// TwinCAT 3 PLC project EcLib
// ProgramVersion: 3.1.4023.0
// libraries:
//   Tc2_Standard, * (Beckhoff Automation GmbH)
//   Tc2_System, * (Beckhoff Automation GmbH)
//   Tc3_Module, * (Beckhoff Automation GmbH)
// project tree:
//   / PlcTask.TcTTO
//   POUs/ MAIN.TcPOU
//   Tasks/ EcMasterConfDevices.TcPOU, EcMasterDeviceCount.TcPOU, EcMasterDeviceState.TcPOU, EcMasterFrameCount.TcPOU, EcMasterFrameStats.TcPOU, EcMasterGetAbnortalStateChange.TcPOU, EcMasterGetDeviceCRC.TcPOU, EcMasterGetDeviceId.TcPOU, EcMasterGetDeviceState.TcPOU, EcMasterProtocolError.TcPOU, EcMasterScanDevices.TcPOU, EcMasterState.TcPOU, IEcTask.TcIO, ITask.TcIO

CONFIGURATION EcLib
    RESOURCE PLC ON TwinCAT3
        TASK PlcTask(INTERVAL := T#10ms, PRIORITY := 20);
        PROGRAM MAIN WITH PlcTask : MAIN;
    END_RESOURCE
END_CONFIGURATION

// ---- Tasks/IEcTask.TcIO
INTERFACE IEcTask EXTENDS ITask

PROPERTY NetID : amsnetid
GET
END_GET
SET
END_SET
END_PROPERTY

END_INTERFACE

// ---- Tasks/ITask.TcIO
INTERFACE ITask

METHOD Abort : BOOL
VAR_INPUT
END_VAR
END_METHOD

PROPERTY Busy : bool
GET
END_GET
END_PROPERTY

PROPERTY Done : bool
GET
END_GET
END_PROPERTY

PROPERTY Error : bool
GET
END_GET
END_PROPERTY

METHOD Execute : BOOL
VAR_INPUT
END_VAR
END_METHOD

END_INTERFACE

// ---- POUs/MAIN.TcPOU
PROGRAM MAIN
VAR
END_VAR

END_PROGRAM

// ---- Tasks/EcMasterConfDevices.TcPOU
FUNCTION_BLOCK EcMasterConfDevices IMPLEMENTS IEcTask
VAR_INPUT
END_VAR
VAR_OUTPUT
END_VAR
VAR
	iState : INT;
	masterConfDevices : Tc2_EtherCAT.FB_EcGetConfSlaves;
	_confDevices : ARRAY[0..Tc2_EtherCAT.EC_MAX_SLAVES] OF Tc2_EtherCAT.ST_EcSlaveConfigData;
	_execute: BOOL;
	_done: BOOL;
	_busy: BOOL;	
	_error: BOOL;
	_netId: AMSNETID;
END_VAR

CASE iState OF
	0:
		IF _execute THEN
			_done := FALSE;
			_busy := TRUE;
			_error := FALSE;
			masterConfDevices.bExecute := TRUE;
			IF masterConfDevices.bBusy THEN
				iState := 10;
				_execute := FALSE;
			END_IF
		END_IF
	10:
		IF NOT masterConfDevices.bBusy THEN
			IF NOT masterConfDevices.bError THEN
				_done := TRUE;
			ELSE
				_error := TRUE;
			END_IF
			_busy := FALSE;
			masterConfDevices.bExecute := FALSE;
			iState := 0;
		END_IF
END_CASE

masterConfDevices(sNetId := Tc2_System.F_CreateAmsNetId(nIds := NetId), 
					pArrEcConfSlaveInfo := ADR(_confDevices), 
					cbBufLen := SIZEOF(_confDevices));

{warning 'add method implementation '}
METHOD Abort : BOOL
masterConfDevices.bExecute := FALSE;
_busy := FALSE;
_execute := FALSE;
Abort := TRUE;
iState := 0;
END_METHOD

{warning 'add property implementation'}
PROPERTY Busy : BOOL
GET
Busy := _busy;
END_GET
END_PROPERTY

PROPERTY ConfiguredDevices : reference to array[0..Ec_Max_slaves] of St_ecslaveconfigdata
GET
ConfiguredDevices REF= _confDevices;
END_GET
END_PROPERTY

{warning 'add property implementation'}
PROPERTY Done : BOOL
GET
Done := _done;
END_GET
END_PROPERTY

{warning 'add property implementation'}
PROPERTY Error : BOOL
GET
Error := _error;
END_GET
END_PROPERTY

{warning 'add method implementation '}
METHOD Execute : BOOL
IF NOT masterConfDevices.bBusy THEN
	Execute := _execute := true;
END_IF
END_METHOD

{warning 'add property implementation'}
PROPERTY NetID : amsnetid
GET
NetID := _netId;
END_GET
SET
_netId := NetID;
END_SET
END_PROPERTY

PROPERTY NumberConfDevices : udint
GET
NumberConfDevices := masterConfDevices.nSlaves;
END_GET
END_PROPERTY

END_FUNCTION_BLOCK

// ---- Tasks/EcMasterDeviceCount.TcPOU
FUNCTION_BLOCK PUBLIC EcMasterDeviceCount IMPLEMENTS IEcTask
VAR_INPUT
END_VAR
VAR_OUTPUT
END_VAR
VAR
	iState : INT;
	masterDeviceCount : Tc2_EtherCAT.FB_EcGetSlaveCount;
	_execute: BOOL;
	_done: BOOL;
	_busy: BOOL;
	_error: BOOL;
	_netId: AMSNETID;
END_VAR

CASE iState OF
	0:
		IF _execute THEN
			_done := FALSE;
			_busy := TRUE;
			_error := FALSE;
			masterDeviceCount.bExecute := TRUE;
			IF masterDeviceCount.bBusy THEN
				iState := 10;
				_execute := false;
			END_IF
		END_IF
	10:
		IF NOT masterDeviceCount.bBusy THEN
			IF NOT masterDeviceCount.bError THEN
				_done := TRUE;
			ELSE
				_error := TRUE;
			END_IF
			_busy := FALSE;
			masterDeviceCount.bExecute := FALSE;
			iState := 0;
		END_IF
END_CASE

masterDeviceCount(sNetId := Tc2_System.F_CreateAmsNetId(nIds := NetId));

{warning 'add method implementation '}
METHOD Abort : BOOL
masterDeviceCount.bExecute := FALSE;
_busy := FALSE;
_execute := FALSE;
Abort := TRUE;
iState := 0;
END_METHOD

{warning 'add property implementation'}
PROPERTY Busy : BOOL
GET
Busy := _busy;
END_GET
END_PROPERTY

{warning 'add property implementation'}
PROPERTY Done : BOOL
GET
Done := _done;
END_GET
END_PROPERTY

{warning 'add property implementation'}
PROPERTY Error : BOOL
GET
Error := _error;
END_GET
END_PROPERTY

METHOD Execute : BOOL
VAR_INPUT
END_VAR
IF NOT Busy THEN
	Execute := _execute := TRUE;
END_IF
END_METHOD

{warning 'add property implementation'}
PROPERTY NetID : amsnetid
GET
NetID := _netId;
END_GET
SET
_netId := NetID;
END_SET
END_PROPERTY

PROPERTY NumberDevices : uint
GET
NumberDevices := masterDeviceCount.nSlaves;
END_GET
END_PROPERTY

END_FUNCTION_BLOCK

// ---- Tasks/EcMasterDeviceState.TcPOU
FUNCTION_BLOCK EcMasterDeviceState IMPLEMENTS IEcTask
VAR_INPUT
END_VAR
VAR_OUTPUT
END_VAR
VAR
	iState : INT;
	masterDeviceState : Tc2_EtherCAT.FB_EcGetMasterDevState;
	_execute: BOOL;
	_done: BOOL;
	_busy: BOOL;
	_error: BOOL;
	_netId: AMSNETID;
END_VAR

CASE iState OF
	0:
		IF _execute THEN
			_done := FALSE;
			_busy := TRUE;
			_error := FALSE;
			masterDeviceState.bExecute := TRUE;
			IF masterDeviceState.bBusy THEN
				iState := 10;
				_execute := false;
			END_IF
		END_IF
	10:
		IF NOT masterDeviceState.bBusy THEN
			IF NOT masterDeviceState.bError THEN
				_done := TRUE;
			ELSE
				_error := TRUE;
			END_IF
			_busy := FALSE;
			masterDeviceState.bExecute := FALSE;
			iState := 0;
		END_IF
END_CASE

masterDeviceState(sNetId := Tc2_System.F_CreateAmsNetId(nIds := NetId));

{warning 'add method implementation '}
METHOD Abort : BOOL
masterDeviceState.bExecute := FALSE;
_busy := FALSE;
_execute := FALSE;
Abort := TRUE;
iState := 0;
END_METHOD

{warning 'add property implementation'}
PROPERTY Busy : BOOL
GET
Busy := _busy;
END_GET
END_PROPERTY

{warning 'add property implementation'}
PROPERTY Done : BOOL
GET
Done := _done;
END_GET
END_PROPERTY

{warning 'add property implementation'}
PROPERTY Error : BOOL
GET
Error := _error;
END_GET
END_PROPERTY

{warning 'add method implementation '}
METHOD Execute : BOOL
IF NOT masterDeviceState.bBusy THEN
	Execute := _execute := true;
END_IF
END_METHOD

PROPERTY MasterDevState : word
GET
MasterDevState := masterDeviceState.nDevState;
END_GET
END_PROPERTY

{warning 'add property implementation'}
PROPERTY NetID : amsnetid
GET
NetID := _netId;
END_GET
SET
_netId := NetID;
END_SET
END_PROPERTY

END_FUNCTION_BLOCK

// ---- Tasks/EcMasterFrameCount.TcPOU
FUNCTION_BLOCK EcMasterFrameCount IMPLEMENTS IEcTask
VAR_INPUT
END_VAR
VAR_OUTPUT
END_VAR
VAR
	iState : INT;
	masterFrameCount : Tc2_EtherCAT.FB_EcMasterFrameCount;
	_execute: BOOL;
	_done: BOOL;
	_busy: BOOL;
	_error: BOOL;
	_netId: AMSNETID;
END_VAR

CASE iState OF
	0:
		IF _execute THEN
			_done := FALSE;
			_busy := TRUE;
			_error := FALSE;
			masterFrameCount.bExecute := TRUE;
			IF masterFrameCount.bBusy THEN
				iState := 10;
				_execute := false;
			END_IF
		END_IF
	10:
		IF NOT masterFrameCount.bBusy THEN
			IF NOT masterFrameCount.bError THEN
				_done := TRUE;
			ELSE
				_error := TRUE;
			END_IF
			_busy := FALSE;
			masterFrameCount.bExecute := FALSE;
			iState := 0;
		END_IF
END_CASE

masterFrameCount(sNetId := Tc2_System.F_CreateAmsNetId(nIds := NetId));

{warning 'add method implementation '}
METHOD Abort : BOOL
masterFrameCount.bExecute := FALSE;
_busy := FALSE;
_execute := FALSE;
Abort := TRUE;
iState := 0;
END_METHOD

{warning 'add property implementation'}
PROPERTY Busy : BOOL
GET
Busy := _busy;
END_GET
END_PROPERTY

{warning 'add property implementation'}
PROPERTY Done : BOOL
GET
Done := _done;
END_GET
END_PROPERTY

{warning 'add property implementation'}
PROPERTY Error : BOOL
GET
Error := _error;
END_GET
END_PROPERTY

{warning 'add method implementation '}
METHOD Execute : BOOL
IF NOT masterFrameCount.bBusy THEN
	Execute := _execute := True;
END_IF
END_METHOD

PROPERTY FrameNumber : UDINT
GET
FrameNumber := masterFrameCount.nFrames;
END_GET
END_PROPERTY

{warning 'add property implementation'}
PROPERTY NetID : amsnetid
GET
NetID := _netId;
END_GET
SET
_netId := NetID;
END_SET
END_PROPERTY

END_FUNCTION_BLOCK

// ---- Tasks/EcMasterFrameStats.TcPOU
FUNCTION_BLOCK PUBLIC EcMasterFrameStats IMPLEMENTS IEcTask
VAR_INPUT
END_VAR
VAR_OUTPUT
END_VAR
VAR
	iState : INT;
	masterFrameStats : Tc2_EtherCAT.FB_EcMasterFrameStatistic;
	_execute: BOOL;
	_done: BOOL;
	_busy: BOOL;
	_error: BOOL;
	_netId: AMSNETID;
END_VAR

CASE iState OF
	0:
		IF _execute THEN
			_done := FALSE;
			_busy := TRUE;
			_error := FALSE;
			masterFrameStats.bExecute := TRUE;
			IF masterFrameStats.bBusy THEN
				iState := 10;
				_execute := false;
			END_IF
		END_IF
	10:
		IF NOT masterFrameStats.bBusy THEN
			IF NOT masterFrameStats.bError THEN
				_done := TRUE;
			ELSE
				_error := TRUE;
			END_IF
			_busy := FALSE;
			masterFrameStats.bExecute := FALSE;
			iState := 0;
		END_IF
END_CASE

masterFrameStats(sNetId := Tc2_System.F_CreateAmsNetId(nIds := NetId));

{warning 'add method implementation '}
METHOD Abort : BOOL
masterFrameStats.bExecute := FALSE;
_busy := FALSE;
_execute := FALSE;
Abort := TRUE;
iState := 0;
END_METHOD

{warning 'add property implementation'}
PROPERTY Busy : BOOL
GET
Busy := _busy;
END_GET
END_PROPERTY

{warning 'add property implementation'}
PROPERTY Done : BOOL
GET
Done := _done;
END_GET
END_PROPERTY

{warning 'add property implementation'}
PROPERTY Error : BOOL
GET
Error := _error;
END_GET
END_PROPERTY

METHOD Execute : BOOL
VAR_INPUT
END_VAR
IF NOT Busy THEN
	Execute := _execute := TRUE;
END_IF
END_METHOD

PROPERTY FramesPerSecond  : LREAL
GET
FramesPerSecond := masterFrameStats.fFramesPerSecond;
END_GET
END_PROPERTY

PROPERTY LostFrames : UDINT
GET
LostFrames := masterFrameStats.nLostFrames;
END_GET
END_PROPERTY

PROPERTY LostQueuedFrames : udint
GET
LostQueuedFrames := masterFrameStats.nLostQueuedFrames;
END_GET
END_PROPERTY

{warning 'add property implementation'}
PROPERTY NetID : amsnetid
GET
NetID := _netId;
END_GET
SET
_netId := NetID;
END_SET
END_PROPERTY

PROPERTY QueuedFramesPerSecond : lreal
GET
QueuedFramesPerSecond := masterFrameStats.fQueuedFramesPerSecond;
END_GET
END_PROPERTY

END_FUNCTION_BLOCK

// ---- Tasks/EcMasterGetAbnortalStateChange.TcPOU
FUNCTION_BLOCK EcMasterGetAbnortalStateChange IMPLEMENTS IEcTask
VAR_INPUT
END_VAR
VAR_OUTPUT
END_VAR
VAR
	iState : INT;
	masterAbnormalStateChanges : Tc2_EtherCAT.FB_EcGetAllSlaveAbnormalStateChanges;
	_abnormalStates : ARRAY[0..Tc2_EtherCAT.EC_MAX_SLAVES] OF UDINT;
	_execute: BOOL;
	_done: BOOL;
	_busy: BOOL;
	_error: BOOL;
	_netId: AMSNETID;
END_VAR

CASE iState OF
	0:
		IF _execute THEN
			_done := FALSE;
			_busy := TRUE;
			_error := FALSE;
			masterAbnormalStateChanges.bExecute := TRUE;
			IF masterAbnormalStateChanges.bBusy THEN
				iState := 10;
				_execute := false;
			END_IF
		END_IF
	10:
		IF NOT masterAbnormalStateChanges.bBusy THEN
			IF NOT masterAbnormalStateChanges.bError THEN
				_done := TRUE;
			ELSE
				_error := TRUE;
			END_IF
			_busy := FALSE;
			masterAbnormalStateChanges.bExecute := FALSE;
			iState := 0;
		END_IF
END_CASE

masterAbnormalStateChanges(sNetId := Tc2_System.F_CreateAmsNetId(nIds := NetId),
							pAddrBuf := ADR(_abnormalStates),
							cbBufLen := SIZEOF(_abnormalStates));

PROPERTY AbnormalStateChanges : reference to array[0..EC_MAX_Slaves] of udint
GET
AbnormalStateChanges REF= _abnormalStates;
END_GET
END_PROPERTY

{warning 'add method implementation '}
METHOD Abort : BOOL
masterAbnormalStateChanges.bExecute := FALSE;
_busy := FALSE;
_execute := FALSE;
Abort := TRUE;
iState := 0;
END_METHOD

{warning 'add property implementation'}
PROPERTY Busy : BOOL
GET
Busy := _busy;
END_GET
END_PROPERTY

{warning 'add property implementation'}
PROPERTY Done : BOOL
GET
Done := _done;
END_GET
END_PROPERTY

{warning 'add property implementation'}
PROPERTY Error : BOOL
GET
Error := _error;
END_GET
END_PROPERTY

{warning 'add method implementation '}
METHOD Execute : BOOL
IF NOT masterAbnormalStateChanges.bBusy THEN
	Execute := _execute := true;
END_IF
END_METHOD

{warning 'add property implementation'}
PROPERTY NetID : amsnetid
GET
NetID := _netId;
END_GET
SET
_netId := NetID;
END_SET
END_PROPERTY

END_FUNCTION_BLOCK

// ---- Tasks/EcMasterGetDeviceCRC.TcPOU
FUNCTION_BLOCK EcMasterGetDeviceCRC IMPLEMENTS IEcTask
VAR_INPUT
END_VAR
VAR_OUTPUT
END_VAR
VAR
	iState : INT;
	getDeviceCRC : Tc2_EtherCAT.FB_EcGetSlaveCrcErrorEx;
	_execute: BOOL;
	_done: BOOL;
	_busy: BOOL;
	_error: BOOL;
	_netId: AMSNETID;
END_VAR

CASE iState OF
	0:
		IF _execute THEN
			_done := FALSE;
			_busy := TRUE;
			_error := FALSE;
			getDeviceCRC.bExecute := TRUE;
			IF getDeviceCRC.bBusy THEN
				iState := 10;
				_execute := false;
			END_IF
		END_IF
	10:
		IF NOT getDeviceCRC.bBusy THEN
			IF NOT getDeviceCRC.bError THEN
				_done := TRUE;
			ELSE
				_error := TRUE;
			END_IF
			_busy := FALSE;
			getDeviceCRC.bExecute := FALSE;
			iState := 0;
		END_IF
END_CASE

getDeviceCRC(sNetId := Tc2_System.F_CreateAmsNetId(nIds := NetId));

{warning 'add method implementation '}
METHOD Abort : BOOL
getDeviceCRC.bExecute := FALSE;
_busy := FALSE;
_execute := FALSE;
Abort := TRUE;
iState := 0;
END_METHOD

{warning 'add property implementation'}
PROPERTY Busy : BOOL
GET
Busy := _busy;
END_GET
END_PROPERTY

PROPERTY DeviceAddr : uint
GET
DeviceAddr := getDeviceCRC.nSlaveAddr;
END_GET
SET
getDeviceCRC.nSlaveAddr := DeviceAddr;
END_SET
END_PROPERTY

PROPERTY DeviceCRC :  ST_EcCrcErrorEx
GET
DeviceCRC := getDeviceCRC.crcError;
END_GET
END_PROPERTY

{warning 'add property implementation'}
PROPERTY Done : BOOL
GET
Done := _done;
END_GET
END_PROPERTY

{warning 'add property implementation'}
PROPERTY Error : BOOL
GET
Error := _error;
END_GET
END_PROPERTY

{warning 'add method implementation '}
METHOD Execute : BOOL
IF NOT getDeviceCRC.bBusy THEN
	Execute := _execute := true;
END_IF
END_METHOD

{warning 'add property implementation'}
PROPERTY NetID : amsnetid
GET
NetID := _netId;
END_GET
SET
_netId := NetID;
END_SET
END_PROPERTY

END_FUNCTION_BLOCK

// ---- Tasks/EcMasterGetDeviceId.TcPOU
FUNCTION_BLOCK EcMasterGetDeviceId IMPLEMENTS IEcTask
VAR_INPUT
END_VAR
VAR_OUTPUT
END_VAR
VAR
	iState : INT;
	getDeviceIdentity : Tc2_EtherCAT.FB_EcGetSlaveIdentity;
	_execute: BOOL;
	_done: BOOL;
	_busy: BOOL;
	_error: BOOL;
	_netId: AMSNETID;
END_VAR

CASE iState OF
	0:
		IF _execute THEN
			_done := FALSE;
			_busy := TRUE;
			_error := FALSE;
			getDeviceIdentity.bExecute := TRUE;
			IF getDeviceIdentity.bBusy THEN
				iState := 10;
				_execute := false;
			END_IF
		END_IF
	10:
		IF NOT getDeviceIdentity.bBusy THEN
			IF NOT getDeviceIdentity.bError THEN
				_done := TRUE;
			ELSE
				_error := TRUE;
			END_IF
			_busy := FALSE;
			getDeviceIdentity.bExecute := FALSE;
			iState := 0;
		END_IF
END_CASE

getDeviceIdentity(sNetId := Tc2_System.F_CreateAmsNetId(nIds := NetId));

{warning 'add method implementation '}
METHOD Abort : BOOL
getDeviceIdentity.bExecute := FALSE;
_busy := FALSE;
_execute := FALSE;
Abort := TRUE;
iState := 0;
END_METHOD

{warning 'add property implementation'}
PROPERTY Busy : BOOL
GET
Busy := _busy;
END_GET
END_PROPERTY

PROPERTY DeviceAddr : uint
GET
DeviceAddr := getDeviceIdentity.nSlaveAddr;
END_GET
SET
getDeviceIdentity.nSlaveAddr := DeviceAddr;
END_SET
END_PROPERTY

PROPERTY DeviceIdentity : ST_EcSlaveIdentity
GET
DeviceIdentity := getDeviceIdentity.identity;
END_GET
END_PROPERTY

{warning 'add property implementation'}
PROPERTY Done : BOOL
GET
Done := _done;
END_GET
END_PROPERTY

{warning 'add property implementation'}
PROPERTY Error : BOOL
GET
Error := _error;
END_GET
END_PROPERTY

{warning 'add method implementation '}
METHOD Execute : BOOL
IF NOT getDeviceIdentity.bBusy THEN
	Execute := _execute := true;
END_IF
END_METHOD

{warning 'add property implementation'}
PROPERTY NetID : amsnetid
GET
NetID := _netId;
END_GET
SET
_netId := NetID;
END_SET
END_PROPERTY

END_FUNCTION_BLOCK

// ---- Tasks/EcMasterGetDeviceState.TcPOU
FUNCTION_BLOCK EcMasterGetDeviceState IMPLEMENTS IEcTask
VAR_INPUT
END_VAR
VAR_OUTPUT
END_VAR
VAR
	iState : INT;
	getDeviceState : Tc2_EtherCAT.FB_EcGetSlaveState;
	_execute: BOOL;
	_done: BOOL;
	_busy: BOOL;
	_error: BOOL;
	_netId: AMSNETID;
END_VAR

CASE iState OF
	0:
		IF _execute THEN
			_done := FALSE;
			_busy := TRUE;
			_error := FALSE;
			getDeviceState.bExecute := TRUE;
			IF getDeviceState.bBusy THEN
				iState := 10;
				_execute := false;
			END_IF
		END_IF
	10:
		IF NOT getDeviceState.bBusy THEN
			IF NOT getDeviceState.bError THEN
				_done := TRUE;
			ELSE
				_error := TRUE;
			END_IF
			_busy := FALSE;
			getDeviceState.bExecute := FALSE;
			iState := 0;
		END_IF
END_CASE

getDeviceState(sNetId := Tc2_System.F_CreateAmsNetId(nIds := NetId));

{warning 'add method implementation '}
METHOD Abort : BOOL
getDeviceState.bExecute := FALSE;
_busy := FALSE;
_execute := FALSE;
Abort := TRUE;
iState := 0;
END_METHOD

{warning 'add property implementation'}
PROPERTY Busy : BOOL
GET
Busy := _busy;
END_GET
END_PROPERTY

PROPERTY DeviceAddr : uint
GET
DeviceAddr := getDeviceState.nSlaveAddr;
END_GET
SET
getDeviceState.nSlaveAddr := DeviceAddr;
END_SET
END_PROPERTY

PROPERTY DeviceState : ST_EcSlaveState
GET
DeviceState := getDeviceState.state;
END_GET
END_PROPERTY

{warning 'add property implementation'}
PROPERTY Done : BOOL
GET
Done := _done;
END_GET
END_PROPERTY

{warning 'add property implementation'}
PROPERTY Error : BOOL
GET
Error := _error;
END_GET
END_PROPERTY

{warning 'add method implementation '}
METHOD Execute : BOOL
IF NOT getDeviceState.bBusy THEN
	Execute := _execute := true;
END_IF
END_METHOD

{warning 'add property implementation'}
PROPERTY NetID : amsnetid
GET
NetID := _netId;
END_GET
SET
_netId := NetID;
END_SET
END_PROPERTY

END_FUNCTION_BLOCK

// ---- Tasks/EcMasterProtocolError.TcPOU
FUNCTION_BLOCK EcMasterProtocolError IMPLEMENTS IEcTask
VAR_INPUT
END_VAR
VAR_OUTPUT
END_VAR
VAR
	iState : INT;
	masterProtocolErr : Tc2_EtherCAT.FB_EcGetLastProtErrInfo;
	_execute: BOOL;
	_done: BOOL;
	_busy: BOOL;
	_error: BOOL;
	_netId: AMSNETID;
END_VAR

CASE iState OF
	0:
		IF _execute THEN
			_done := FALSE;
			_busy := TRUE;
			_error := FALSE;
			masterProtocolErr.bExecute := TRUE;
			IF masterProtocolErr.bBusy THEN
				iState := 10;
				_execute := false;
			END_IF
		END_IF
	10:
		IF NOT masterProtocolErr.bBusy THEN
			IF NOT masterProtocolErr.bError THEN
				_done := TRUE;
			ELSE
				_error := TRUE;
			END_IF
			_busy := FALSE;
			masterProtocolErr.bExecute := FALSE;
			iState := 0;
		END_IF
END_CASE

masterProtocolErr(sNetId := Tc2_System.F_CreateAmsNetId(nIds := NetId));

{warning 'add method implementation '}
METHOD Abort : BOOL
masterProtocolErr.bExecute := FALSE;
_busy := FALSE;
_execute := FALSE;
Abort := TRUE;
iState := 0;
END_METHOD

{warning 'add property implementation'}
PROPERTY Busy : BOOL
GET
Busy := _busy;
END_GET
END_PROPERTY

PROPERTY DeviceAddr : uint
GET
DeviceAddr := masterProtocolErr.nSlaveAddr;
END_GET
SET
masterProtocolErr.nSlaveAddr := DeviceAddr;
END_SET
END_PROPERTY

{warning 'add property implementation'}
PROPERTY Done : BOOL
GET
Done := _done;
END_GET
END_PROPERTY

{warning 'add property implementation'}
PROPERTY Error : BOOL
GET
Error := _error;
END_GET
END_PROPERTY

{warning 'add method implementation '}
METHOD Execute : BOOL
IF NOT masterProtocolErr.bBusy THEN
	Execute := _execute := TRUE;
END_IF
END_METHOD

PROPERTY LastProtocolError : ST_EcLastProtErrInfo
GET
LastProtocolError := masterProtocolErr.info;
END_GET
END_PROPERTY

{warning 'add property implementation'}
PROPERTY NetID : amsnetid
GET
NetID := _netId;
END_GET
SET
_netId := NetID;
END_SET
END_PROPERTY

PROPERTY ProtocolType : E_EcMbxProtType
GET
ProtocolType := masterProtocolErr.eProtocol;
END_GET
SET
masterProtocolErr.eProtocol := ProtocolType;
END_SET
END_PROPERTY

END_FUNCTION_BLOCK

// ---- Tasks/EcMasterScanDevices.TcPOU
FUNCTION_BLOCK EcMasterScanDevices IMPLEMENTS IEcTask
VAR_INPUT
END_VAR
VAR_OUTPUT
END_VAR
VAR
	iState : INT;
	masterScanDevices : Tc2_EtherCAT.FB_EcGetScannedSlaves;
	_scanDevices : ARRAY[0..Tc2_EtherCAT.EC_MAX_SLAVES] OF Tc2_EtherCAT.ST_EcSlaveScannedData;
	_execute: BOOL;
	_done: BOOL;
	_busy: BOOL;
	_error: BOOL;
	_netId: AMSNETID;
END_VAR

CASE iState OF
	0:
		IF _execute THEN
			_done := FALSE;
			_busy := TRUE;
			_error := FALSE;
			masterScanDevices.bExecute := TRUE;
			IF masterScanDevices.bBusy THEN
				iState := 10;
				_execute := false;
			END_IF
		END_IF
	10:
		IF NOT masterScanDevices.bBusy THEN
			IF NOT masterScanDevices.bError THEN
				_done := TRUE;
			ELSE
				_error := TRUE;
			END_IF
			_busy := FALSE;
			masterScanDevices.bExecute := FALSE;
			iState := 0;
		END_IF
END_CASE

masterScanDevices(sNetId := Tc2_System.F_CreateAmsNetId(nIds := NetId), 
					pArrEcScannedSlaveInfo := ADR(_scanDevices), 
					cbBufLen := SIZEOF(_scanDevices));

{warning 'add method implementation '}
METHOD Abort : BOOL
masterScanDevices.bExecute := FALSE;
_busy := FALSE;
_execute := FALSE;
Abort := TRUE;
iState := 0;
END_METHOD

{warning 'add property implementation'}
PROPERTY Busy : BOOL
GET
Busy := _busy;
END_GET
END_PROPERTY

{warning 'add property implementation'}
PROPERTY Done : BOOL
GET
Done := _done;
END_GET
END_PROPERTY

{warning 'add property implementation'}
PROPERTY Error : BOOL
GET
Error := _error;
END_GET
END_PROPERTY

{warning 'add method implementation '}
METHOD Execute : BOOL
IF NOT masterScanDevices.bBusy THEN
	Execute := _execute := true;
END_IF
END_METHOD

{warning 'add property implementation'}
PROPERTY NetID : amsnetid
GET
NetID := _netId;
END_GET
SET
_netId := NetID;
END_SET
END_PROPERTY

PROPERTY NumberScanDevices : udint
GET
NumberScanDevices := masterScanDevices.nSlaves;
END_GET
END_PROPERTY

PROPERTY ScannedDevices : reference to array[0..EC_MAX_Slaves] of ST_EcSlaveScannedData
GET
ScannedDevices REF= _scanDevices;
END_GET
END_PROPERTY

END_FUNCTION_BLOCK

// ---- Tasks/EcMasterState.TcPOU
{attribute 'hide_all_locals'}
FUNCTION_BLOCK EcMasterState IMPLEMENTS IEcTask
VAR_INPUT
END_VAR
VAR_OUTPUT
END_VAR
VAR
	iState : INT;
	getMasterState : Tc2_EtherCAT.FB_EcGetMasterState;
	_execute: BOOL;
	_done: BOOL;
	_busy: BOOL;
	_error: BOOL;
	
END_VAR

CASE iState OF
	0:
		IF _execute THEN
			_done := FALSE;
			_busy := TRUE;
			_error := FALSE;
			getMasterState.bExecute := TRUE;
			IF getMasterState.bBusy THEN
				iState := 10;
				_execute := false;
			END_IF
		END_IF
	10:
		IF NOT getMasterState.bBusy THEN
			IF NOT getMasterState.bError THEN
				_done := TRUE;
			ELSE
				_error := TRUE;
			END_IF
			_busy := FALSE;
			getMasterState.bExecute := FALSE;
			iState := 0;
		END_IF
END_CASE

getMasterState(sNetId := Tc2_System.F_CreateAmsNetId(nIds := NetId));

{warning 'add method implementation '}
METHOD Abort : BOOL
getMasterState.bExecute := FALSE;
_busy := FALSE;
_execute := FALSE;
Abort := TRUE;
iState := 0;
END_METHOD

{warning 'add property implementation'}
PROPERTY Busy : BOOL
GET
Busy := _busy;
END_GET
END_PROPERTY

{warning 'add property implementation'}
PROPERTY Done : BOOL
GET
Done := _done;
END_GET
END_PROPERTY

{warning 'add property implementation'}
PROPERTY Error : BOOL
GET
Error := _error;
END_GET
END_PROPERTY

{warning 'add method implementation '}
METHOD Execute : BOOL
IF NOT getMasterState.bBusy THEN
	Execute := _execute := TRUE;
END_IF
END_METHOD

PROPERTY MasterState : word
GET
MasterState := getMasterState.state;
END_GET
END_PROPERTY

{warning 'add property implementation'}
PROPERTY NetID : amsnetid
GET
NetID := _netId;
END_GET
SET
_netId := NetID;
END_SET
END_PROPERTY

END_FUNCTION_BLOCK
